(* Logix 5000 project; controller GEA_Test_Chamber vendor 1 type 14 code 196 rev 32.14; software revision 32.04; part 11 of 11 *)
(* tags used below, declared in another part *)
   Mod_Serv_On : BOOL;
   ModbusTCPIP_Data_SWPB : INT[100];
   TC : INT[30];
   always_off : BOOL;
   FVIR_Error_MSG : INT;
   FVIR_LabView_Status : INT;
   FVIR_Rate_REAL : REAL;
   FVIR_Totalizer_REAL : REAL;
   Heater_Cnt : COUNTER;
   LDO_Error_MSG : INT;
   LDO_LabView_Status : INT;
   Modbus_LabView : raC_Opr_NetModbusTCPServer;
   Modbus_LabView_Data : raC_UDT_ModbusServerData;
   Modbus_LabView_EN : BOOL;
   Modbus_LabView_MSG_Accept : MESSAGE;
   Modbus_LabView_MSG_Create : MESSAGE;
   Modbus_LabView_MSG_Delete : MESSAGE;
   Modbus_LabView_MSG_DeleteAll : MESSAGE;
   Modbus_LabView_MSG_Read : MESSAGE;
   Modbus_LabView_MSG_SetSing : MESSAGE;
   Modbus_LabView_MSG_Write : MESSAGE;
   Modbus_LabView_Parameters : raC_UDT_ModbusServerBase;
   nLDO_Rate_REAL : REAL;
   nLDO_Totalizer_REAL : REAL;
   Oil_inj_08_Cnt : COUNTER;
   Oil_inj_11_Cnt : COUNTER;
   Oil_inj_133_Cnt : COUNTER;
(* Modbus_LabView, continued *)

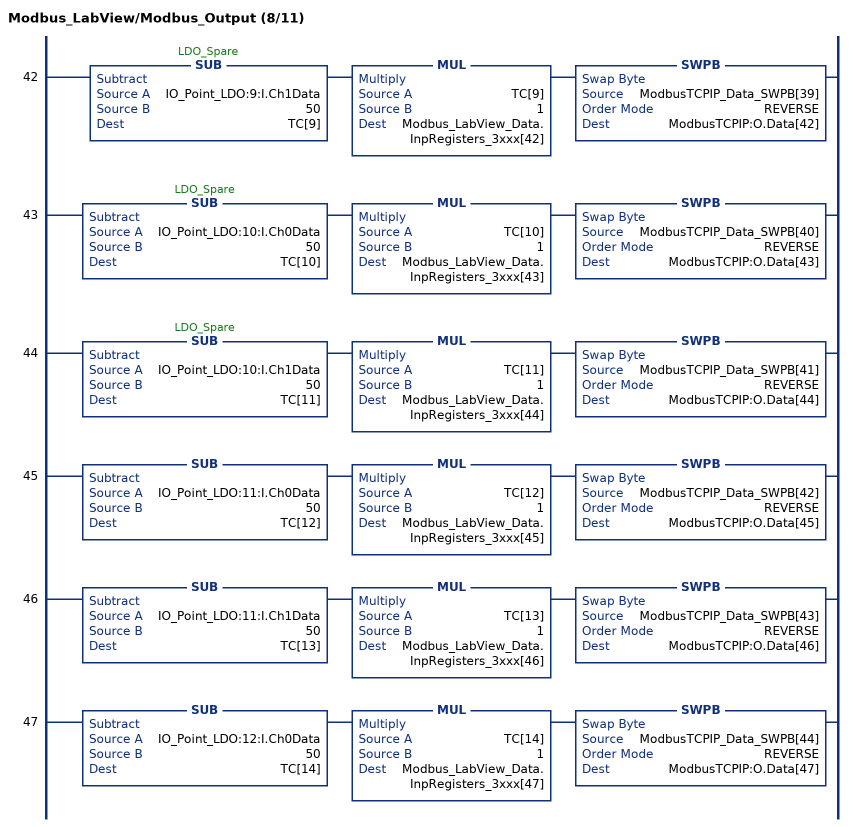
   [picture p213: Modbus_LabView/Modbus_Output rungs 42-47]
   42: SUB(IO_Point_LDO:9:I.Ch1Data,50,TC[9])MUL(TC[9],1,Modbus_LabView_Data.InpRegisters_3xxx[42])SWPB(ModbusTCPIP_Data_SWPB[39],REVERSE,ModbusTCPIP:O.Data[42]);
   43: SUB(IO_Point_LDO:10:I.Ch0Data,50,TC[10])MUL(TC[10],1,Modbus_LabView_Data.InpRegisters_3xxx[43])SWPB(ModbusTCPIP_Data_SWPB[40],REVERSE,ModbusTCPIP:O.Data[43]);
   44: SUB(IO_Point_LDO:10:I.Ch1Data,50,TC[11])MUL(TC[11],1,Modbus_LabView_Data.InpRegisters_3xxx[44])SWPB(ModbusTCPIP_Data_SWPB[41],REVERSE,ModbusTCPIP:O.Data[44]);
   45: SUB(IO_Point_LDO:11:I.Ch0Data,50,TC[12])MUL(TC[12],1,Modbus_LabView_Data.InpRegisters_3xxx[45])SWPB(ModbusTCPIP_Data_SWPB[42],REVERSE,ModbusTCPIP:O.Data[45]);
   46: SUB(IO_Point_LDO:11:I.Ch1Data,50,TC[13])MUL(TC[13],1,Modbus_LabView_Data.InpRegisters_3xxx[46])SWPB(ModbusTCPIP_Data_SWPB[43],REVERSE,ModbusTCPIP:O.Data[46]);
   47: SUB(IO_Point_LDO:12:I.Ch0Data,50,TC[14])MUL(TC[14],1,Modbus_LabView_Data.InpRegisters_3xxx[47])SWPB(ModbusTCPIP_Data_SWPB[44],REVERSE,ModbusTCPIP:O.Data[47]);
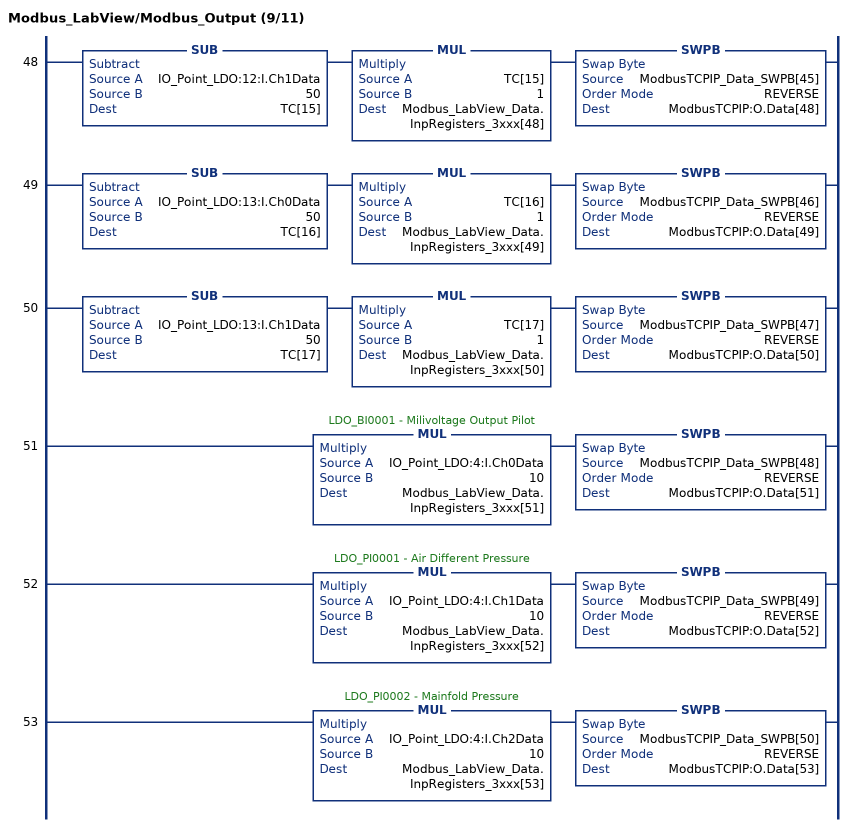
   48: SUB(IO_Point_LDO:12:I.Ch1Data,50,TC[15])MUL(TC[15],1,Modbus_LabView_Data.InpRegisters_3xxx[48])SWPB(ModbusTCPIP_Data_SWPB[45],REVERSE,ModbusTCPIP:O.Data[48]);
   49: SUB(IO_Point_LDO:13:I.Ch0Data,50,TC[16])MUL(TC[16],1,Modbus_LabView_Data.InpRegisters_3xxx[49])SWPB(ModbusTCPIP_Data_SWPB[46],REVERSE,ModbusTCPIP:O.Data[49]);
   50: SUB(IO_Point_LDO:13:I.Ch1Data,50,TC[17])MUL(TC[17],1,Modbus_LabView_Data.InpRegisters_3xxx[50])SWPB(ModbusTCPIP_Data_SWPB[47],REVERSE,ModbusTCPIP:O.Data[50]);
   51: MUL(IO_Point_LDO:4:I.Ch0Data,10,Modbus_LabView_Data.InpRegisters_3xxx[51])SWPB(ModbusTCPIP_Data_SWPB[48],REVERSE,ModbusTCPIP:O.Data[51]);
   52: MUL(IO_Point_LDO:4:I.Ch1Data,10,Modbus_LabView_Data.InpRegisters_3xxx[52])SWPB(ModbusTCPIP_Data_SWPB[49],REVERSE,ModbusTCPIP:O.Data[52]);
   53: MUL(IO_Point_LDO:4:I.Ch2Data,10,Modbus_LabView_Data.InpRegisters_3xxx[53])SWPB(ModbusTCPIP_Data_SWPB[50],REVERSE,ModbusTCPIP:O.Data[53]);
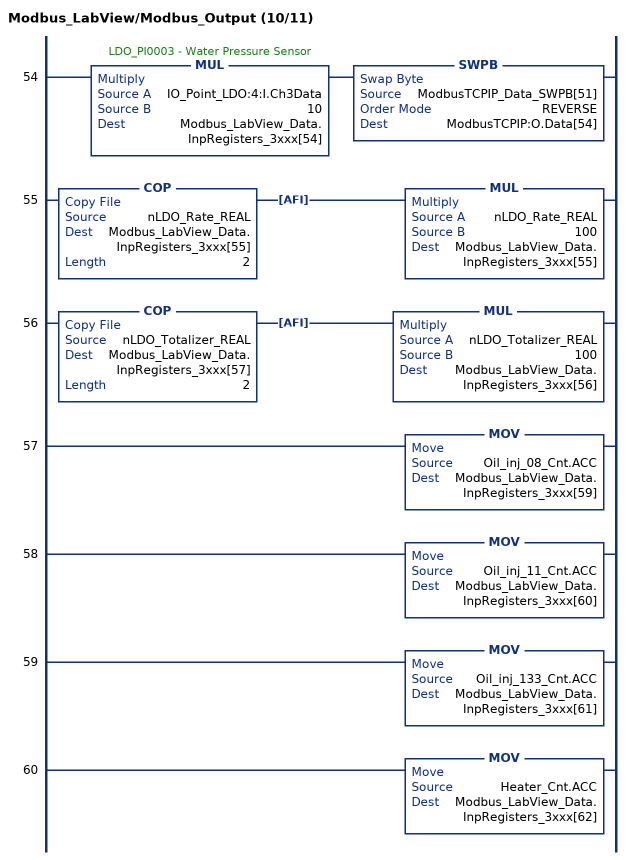
   54: MUL(IO_Point_LDO:4:I.Ch3Data,10,Modbus_LabView_Data.InpRegisters_3xxx[54])SWPB(ModbusTCPIP_Data_SWPB[51],REVERSE,ModbusTCPIP:O.Data[54]);
   55: COP(nLDO_Rate_REAL,Modbus_LabView_Data.InpRegisters_3xxx[55],2)AFI()MUL(nLDO_Rate_REAL,100,Modbus_LabView_Data.InpRegisters_3xxx[55]);
   56: COP(nLDO_Totalizer_REAL,Modbus_LabView_Data.InpRegisters_3xxx[57],2)AFI()MUL(nLDO_Totalizer_REAL,100,Modbus_LabView_Data.InpRegisters_3xxx[56]);
   57: MOV(Oil_inj_08_Cnt.ACC,Modbus_LabView_Data.InpRegisters_3xxx[59]);
   58: MOV(Oil_inj_11_Cnt.ACC,Modbus_LabView_Data.InpRegisters_3xxx[60]);
   59: MOV(Oil_inj_133_Cnt.ACC,Modbus_LabView_Data.InpRegisters_3xxx[61]);
   60: MOV(Heater_Cnt.ACC,Modbus_LabView_Data.InpRegisters_3xxx[62]);
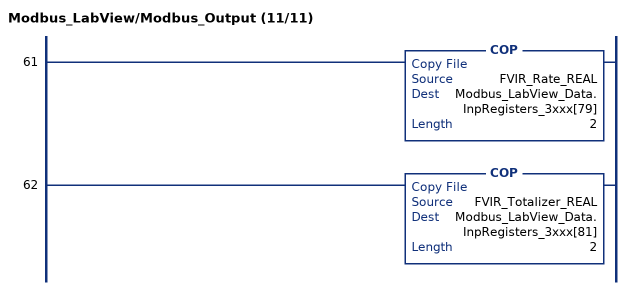
   61: COP(FVIR_Rate_REAL,Modbus_LabView_Data.InpRegisters_3xxx[79],2);
   62: COP(FVIR_Totalizer_REAL,Modbus_LabView_Data.InpRegisters_3xxx[81],2);
END_ROUTINE

ROUTINE Modbus_Server   (* ladder *)
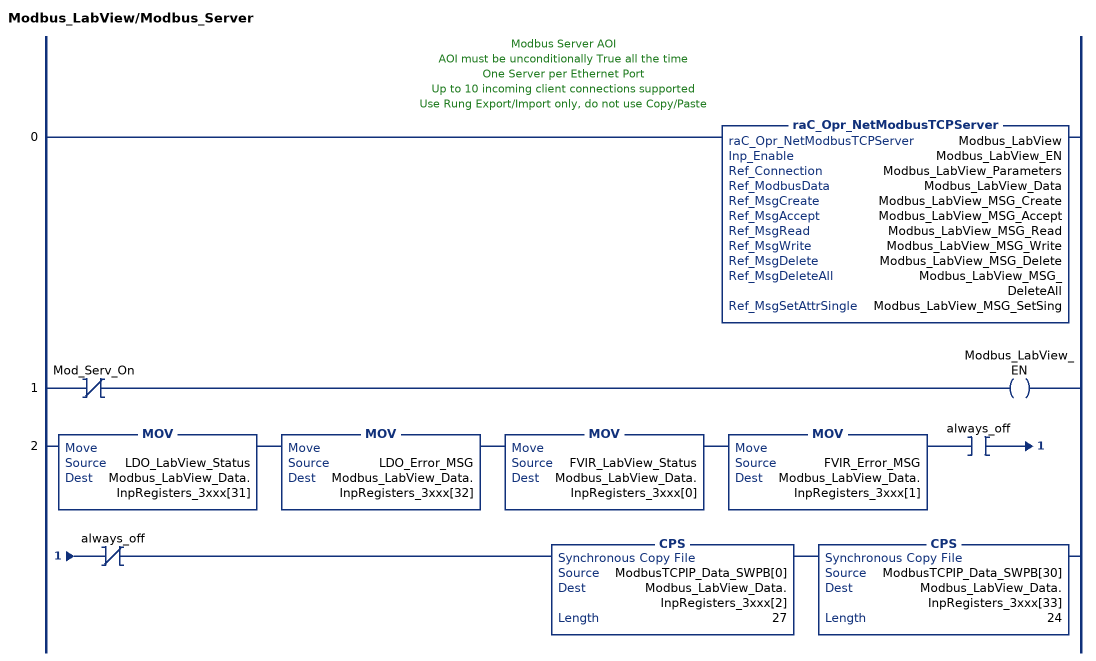
   // Modbus Server AOI
   // AOI must be unconditionally True all the time
   // One Server per Ethernet Port
   // Up to 10 incoming client connections supported
   // Use Rung Export/Import only, do not use Copy/Paste
   0: raC_Opr_NetModbusTCPServer(Modbus_LabView,Modbus_LabView_EN,Modbus_LabView_Parameters,Modbus_LabView_Data,Modbus_LabView_MSG_Create,Modbus_LabView_MSG_Accept,Modbus_LabView_MSG_Read,Modbus_LabView_MSG_Write,Modbus_LabView_MSG_Delete,Modbus_LabView_MSG_DeleteAll,Modbus_LabView_MSG_SetSing);
   1: XIO(Mod_Serv_On)OTE(Modbus_LabView_EN);
   2: MOV(LDO_LabView_Status,Modbus_LabView_Data.InpRegisters_3xxx[31])MOV(LDO_Error_MSG,Modbus_LabView_Data.InpRegisters_3xxx[32])MOV(FVIR_LabView_Status,Modbus_LabView_Data.InpRegisters_3xxx[0])MOV(FVIR_Error_MSG,Modbus_LabView_Data.InpRegisters_3xxx[1])XIC(always_off)XIO(always_off)CPS(ModbusTCPIP_Data_SWPB[0],Modbus_LabView_Data.InpRegisters_3xxx[2],27)CPS(ModbusTCPIP_Data_SWPB[30],Modbus_LabView_Data.InpRegisters_3xxx[33],24);
END_ROUTINE
END_PROGRAM
